// TIA Portal project "Controle_Por_Horario" (V18)

(* hardware
DEVICE "S7-1200 station_1"  S7-1200 Station
   slot 0: "Rack_0"  S7-1200 Rack  Rack  V1.0
   slot 1: "PLC_1"  CPU 1214C DC/DC/DC  6ES7 214-1AG40-0XB0  V4.5
DEVICE "HMI_1"  KTP700 Basic PN
   slot 0: "HMI_1"  KTP700 Basic PN  6AV2 123-2GB03-0AX0  17.0.0.0
   slot 1: "HMI_RT_1"  KTP700 Basic PN  6AV2 123-2GB03-0AX0  17.0.0.0
   slot 5: "HMI_1.IE_CP_1"  PROFINET Interface  17.0.0.0
      slot 1: "PROFINET Interface_1"  PROFINET Interface
         slot 1: "Port_1"  Port
*)

// ===== PLC "PLC_1"  CPU 1214C DC/DC/DC =====

VAR_GLOBAL   // PLC tag table "Default tag table"
   "System_Byte" AT %MB1 : Byte;
   "FirstScan" AT %M1.0 : Bool;
   "DiagStatusUpdate" AT %M1.1 : Bool;
   "AlwaysTRUE" AT %M1.2 : Bool;
   "AlwaysFALSE" AT %M1.3 : Bool;
   "Clock_Byte" AT %MB0 : Byte;
   "Clock_10Hz" AT %M0.0 : Bool;
   "Clock_5Hz" AT %M0.1 : Bool;
   "Clock_2.5Hz" AT %M0.2 : Bool;
   "Clock_2Hz" AT %M0.3 : Bool;
   "Clock_1.25Hz" AT %M0.4 : Bool;
   "Clock_1Hz" AT %M0.5 : Bool;
   "Clock_0.625Hz" AT %M0.6 : Bool;
   "Clock_0.5Hz" AT %M0.7 : Bool;
END_VAR

// folder: DBs

DATA_BLOCK "Var_IHM"   // DB1
{ S7_Optimized_Access := 'TRUE' }
VERSION : 0.1
   VAR
      Tela_Root : Struct
         Int_Date_Time_Local : Int;
         Date_Time_Formated : String;
         Date_Time : DTL;
         Bt_Liga_Habilita_Domingo : Bool;
         Bt_Liga_Habilita_Segunda : Bool;
         Bt_Liga_Habilita_Terca : Bool;
         Bt_Liga_Habilita_Quarta : Bool;
         Bt_Liga_Habilita_Quinta : Bool;
         Bt_Liga_Habilita_Sexta : Bool;
         Bt_Liga_Habilita_Sabado : Bool;
         Hora_Liga_Domingo : USInt;
         Minuto_Liga_Domingo : USInt;
         Hora_Liga_Segunda : USInt;
         Minuto_Liga_Segunda : USInt;
         Hora_Liga_Terca : USInt;
         Minuto_Liga_Terca : USInt;
         Hora_Liga_Quarta : USInt;
         Minuto_Liga_Quarta : USInt;
         Hora_Liga_Quinta : USInt;
         Minuto_Liga_Quinta : USInt;
         Hora_Liga_Sexta : USInt;
         Minuto_Liga_Sexta : USInt;
         Hora_Liga_Sabado : USInt;
         Minuto_Liga_Sabado : USInt;
         Hora_Desliga_Domingo : USInt;
         Minuto_Desliga_Domingo : USInt;
         Hora_Desliga_Segunda : USInt;
         Minuto_Desliga_Segunda : USInt;
         Hora_Desliga_Terca : USInt;
         Minuto_Desliga_Terca : USInt;
         Hora_Desliga_Quarta : USInt;
         Minuto_Desliga_Quarta : USInt;
         Hora_Desliga_Quinta : USInt;
         Minuto_Desliga_Quinta : USInt;
         Hora_Desliga_Sexta : USInt;
         Minuto_Desliga_Sexta : USInt;
         Hora_Desliga_Sabado : USInt;
         Minuto_Desliga_Sabado : USInt;
         Liga : Bool;
      END_STRUCT;
   END_VAR
BEGIN
END_DATA_BLOCK

// folder: (top level)

ORGANIZATION_BLOCK "Main"   // OB1, LAD, ProgramCycle
TITLE = "Main Program Sweep (Cycle)"
{ S7_Optimized_Access := 'TRUE' }
VERSION : 0.1
   VAR_INPUT
      Initial_Call : Bool;   // Initial call of this OB
      Remanence : Bool;   // =True, if remanent data are available
   END_VAR
BEGIN

REGION Network 1
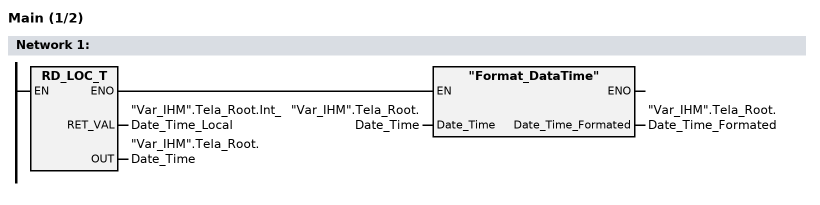
   // ENO of a box is taken as its EN; it also drops when the box reports an error
   "Var_IHM".Tela_Root.Int_Date_Time_Local := RD_LOC_T(OUT => "Var_IHM".Tela_Root.Date_Time);
   "Format_DataTime"(Date_Time := "Var_IHM".Tela_Root.Date_Time,
                     Date_Time_Formated => "Var_IHM".Tela_Root.Date_Time_Formated);
END_REGION

REGION Network 2
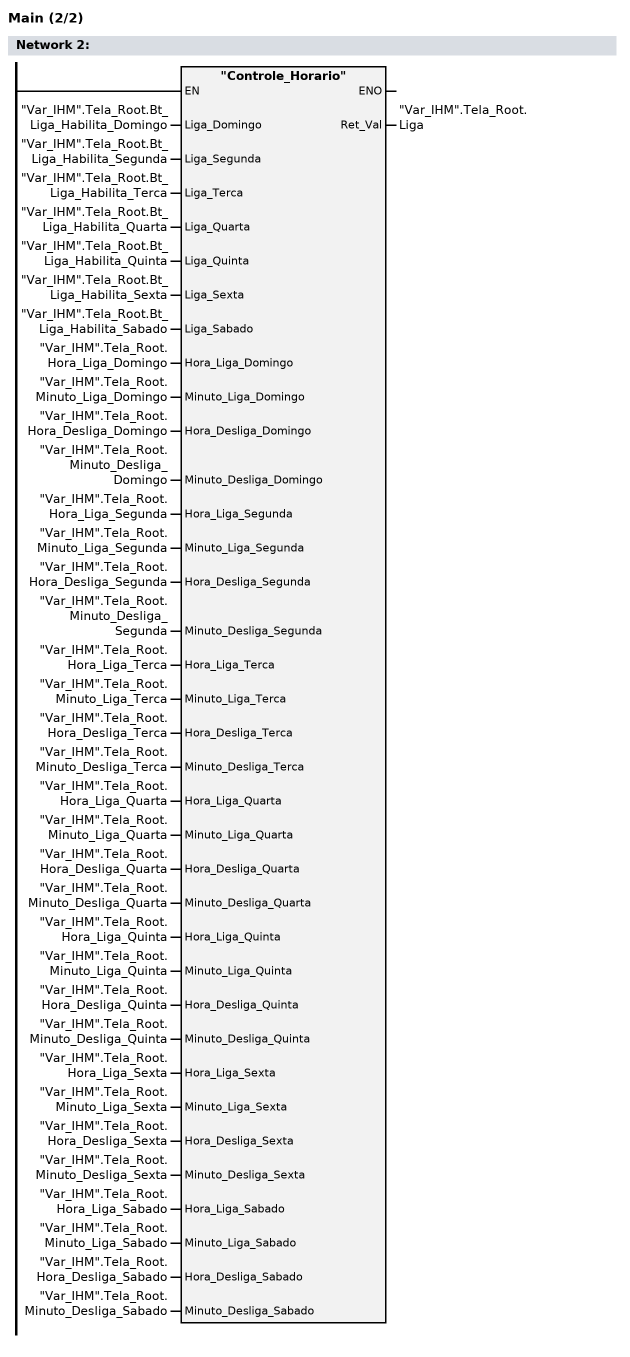
   RUNG wire#powerrail
      "Controle_Horario"(Liga_Domingo := "Var_IHM".Tela_Root.Bt_Liga_Habilita_Domingo, Liga_Segunda := "Var_IHM".Tela_Root.Bt_Liga_Habilita_Segunda, Liga_Terca := "Var_IHM".Tela_Root.Bt_Liga_Habilita_Terca, Liga_Quarta := "Var_IHM".Tela_Root.Bt_Liga_Habilita_Quarta, Liga_Quinta := "Var_IHM".Tela_Root.Bt_Liga_Habilita_Quinta, Liga_Sexta := "Var_IHM".Tela_Root.Bt_Liga_Habilita_Sexta, Liga_Sabado := "Var_IHM".Tela_Root.Bt_Liga_Habilita_Sabado, Hora_Liga_Domingo := "Var_IHM".Tela_Root.Hora_Liga_Domingo, Minuto_Liga_Domingo := "Var_IHM".Tela_Root.Minuto_Liga_Domingo, Hora_Desliga_Domingo := "Var_IHM".Tela_Root.Hora_Desliga_Domingo, Minuto_Desliga_Domingo := "Var_IHM".Tela_Root.Minuto_Desliga_Domingo, Hora_Liga_Segunda := "Var_IHM".Tela_Root.Hora_Liga_Segunda, Minuto_Liga_Segunda := "Var_IHM".Tela_Root.Minuto_Liga_Segunda, Hora_Desliga_Segunda := "Var_IHM".Tela_Root.Hora_Desliga_Segunda, Minuto_Desliga_Segunda := "Var_IHM".Tela_Root.Minuto_Desliga_Segunda, Hora_Liga_Terca := "Var_IHM".Tela_Root.Hora_Liga_Terca, Minuto_Liga_Terca := "Var_IHM".Tela_Root.Minuto_Liga_Terca, Hora_Desliga_Terca := "Var_IHM".Tela_Root.Hora_Desliga_Terca, Minuto_Desliga_Terca := "Var_IHM".Tela_Root.Minuto_Desliga_Terca, Hora_Liga_Quarta := "Var_IHM".Tela_Root.Hora_Liga_Quarta, Minuto_Liga_Quarta := "Var_IHM".Tela_Root.Minuto_Liga_Quarta, Hora_Desliga_Quarta := "Var_IHM".Tela_Root.Hora_Desliga_Quarta, Minuto_Desliga_Quarta := "Var_IHM".Tela_Root.Minuto_Desliga_Quarta, Hora_Liga_Quinta := "Var_IHM".Tela_Root.Hora_Liga_Quinta, Minuto_Liga_Quinta := "Var_IHM".Tela_Root.Minuto_Liga_Quinta, Hora_Desliga_Quinta := "Var_IHM".Tela_Root.Hora_Desliga_Quinta, Minuto_Desliga_Quinta := "Var_IHM".Tela_Root.Minuto_Desliga_Quinta, Hora_Liga_Sexta := "Var_IHM".Tela_Root.Hora_Liga_Sexta, Minuto_Liga_Sexta := "Var_IHM".Tela_Root.Minuto_Liga_Sexta, Hora_Desliga_Sexta := "Var_IHM".Tela_Root.Hora_Desliga_Sexta, Minuto_Desliga_Sexta := "Var_IHM".Tela_Root.Minuto_Desliga_Sexta, Hora_Liga_Sabado := "Var_IHM".Tela_Root.Hora_Liga_Sabado, Minuto_Liga_Sabado := "Var_IHM".Tela_Root.Minuto_Liga_Sabado, Hora_Desliga_Sabado := "Var_IHM".Tela_Root.Hora_Desliga_Sabado, Minuto_Desliga_Sabado := "Var_IHM".Tela_Root.Minuto_Desliga_Sabado, Ret_Val => "Var_IHM".Tela_Root.Liga)
   END_RUNG
   // the same network as SCL:
   "Var_IHM".Tela_Root.Liga := "Controle_Horario"(Liga_Domingo := "Var_IHM".Tela_Root.Bt_Liga_Habilita_Domingo,
                           Liga_Segunda := "Var_IHM".Tela_Root.Bt_Liga_Habilita_Segunda,
                           Liga_Terca := "Var_IHM".Tela_Root.Bt_Liga_Habilita_Terca,
                           Liga_Quarta := "Var_IHM".Tela_Root.Bt_Liga_Habilita_Quarta,
                           Liga_Quinta := "Var_IHM".Tela_Root.Bt_Liga_Habilita_Quinta,
                           Liga_Sexta := "Var_IHM".Tela_Root.Bt_Liga_Habilita_Sexta,
                           Liga_Sabado := "Var_IHM".Tela_Root.Bt_Liga_Habilita_Sabado,
                           Hora_Liga_Domingo := "Var_IHM".Tela_Root.Hora_Liga_Domingo,
                           Minuto_Liga_Domingo := "Var_IHM".Tela_Root.Minuto_Liga_Domingo,
                           Hora_Desliga_Domingo := "Var_IHM".Tela_Root.Hora_Desliga_Domingo,
                           Minuto_Desliga_Domingo := "Var_IHM".Tela_Root.Minuto_Desliga_Domingo,
                           Hora_Liga_Segunda := "Var_IHM".Tela_Root.Hora_Liga_Segunda,
                           Minuto_Liga_Segunda := "Var_IHM".Tela_Root.Minuto_Liga_Segunda,
                           Hora_Desliga_Segunda := "Var_IHM".Tela_Root.Hora_Desliga_Segunda,
                           Minuto_Desliga_Segunda := "Var_IHM".Tela_Root.Minuto_Desliga_Segunda,
                           Hora_Liga_Terca := "Var_IHM".Tela_Root.Hora_Liga_Terca,
                           Minuto_Liga_Terca := "Var_IHM".Tela_Root.Minuto_Liga_Terca,
                           Hora_Desliga_Terca := "Var_IHM".Tela_Root.Hora_Desliga_Terca,
                           Minuto_Desliga_Terca := "Var_IHM".Tela_Root.Minuto_Desliga_Terca,
                           Hora_Liga_Quarta := "Var_IHM".Tela_Root.Hora_Liga_Quarta,
                           Minuto_Liga_Quarta := "Var_IHM".Tela_Root.Minuto_Liga_Quarta,
                           Hora_Desliga_Quarta := "Var_IHM".Tela_Root.Hora_Desliga_Quarta,
                           Minuto_Desliga_Quarta := "Var_IHM".Tela_Root.Minuto_Desliga_Quarta,
                           Hora_Liga_Quinta := "Var_IHM".Tela_Root.Hora_Liga_Quinta,
                           Minuto_Liga_Quinta := "Var_IHM".Tela_Root.Minuto_Liga_Quinta,
                           Hora_Desliga_Quinta := "Var_IHM".Tela_Root.Hora_Desliga_Quinta,
                           Minuto_Desliga_Quinta := "Var_IHM".Tela_Root.Minuto_Desliga_Quinta,
                           Hora_Liga_Sexta := "Var_IHM".Tela_Root.Hora_Liga_Sexta,
                           Minuto_Liga_Sexta := "Var_IHM".Tela_Root.Minuto_Liga_Sexta,
                           Hora_Desliga_Sexta := "Var_IHM".Tela_Root.Hora_Desliga_Sexta,
                           Minuto_Desliga_Sexta := "Var_IHM".Tela_Root.Minuto_Desliga_Sexta,
                           Hora_Liga_Sabado := "Var_IHM".Tela_Root.Hora_Liga_Sabado,
                           Minuto_Liga_Sabado := "Var_IHM".Tela_Root.Minuto_Liga_Sabado,
                           Hora_Desliga_Sabado := "Var_IHM".Tela_Root.Hora_Desliga_Sabado,
                           Minuto_Desliga_Sabado := "Var_IHM".Tela_Root.Minuto_Desliga_Sabado);
END_REGION
END_ORGANIZATION_BLOCK

// folder: FCs

FUNCTION "Format_DataTime" : Void   // FC1, SCL
TITLE = Ezequiel
{ S7_Optimized_Access := 'TRUE' }
VERSION : 0.1
// Formata data e hora para o padrao DD/MM/YYYY  HH:MM:SS
   VAR_INPUT
      Date_Time : DTL;
   END_VAR
   VAR_OUTPUT
      Date_Time_Formated : String;
   END_VAR
   VAR_TEMP
      YEAR : String;
      MONTH : String;
      DAY : String;
      HOUR : String;
      MINUTE : String;
      SECOND : String;
      "DATE" : String;
      "TIME" : String;
   END_VAR
BEGIN
   #YEAR := UINT_TO_STRING(#Date_Time.YEAR);
   #YEAR := RIGHT(IN := #YEAR, L := 4);
   #MONTH := USINT_TO_STRING(#Date_Time.MONTH);

   IF #Date_Time.MONTH >= 10 THEN
       #MONTH := RIGHT(IN := #MONTH, L := 2);
   ELSE
       #MONTH := RIGHT(IN := #MONTH, L := 1);
       #MONTH := CONCAT(IN1 := '0', IN2 := #MONTH);
   END_IF;

   #DAY := USINT_TO_STRING(#Date_Time.DAY);

   IF #Date_Time.DAY >= 10 THEN
       #DAY := RIGHT(IN := #DAY, L := 2);
   ELSE
       #DAY := RIGHT(IN := #DAY, L := 1);
       #DAY := CONCAT(IN1 := '0', IN2 :=#DAY);
   END_IF;


   #HOUR := USINT_TO_STRING(#Date_Time.HOUR);

   IF #Date_Time.HOUR >= 10 THEN
       #HOUR := RIGHT(IN := #HOUR, L := 2);
   ELSE
       #HOUR := RIGHT(IN := #HOUR, L := 1);
   END_IF;

   #MINUTE := USINT_TO_STRING(#Date_Time.MINUTE);

   IF #Date_Time.MINUTE >= 10 THEN
       #MINUTE := RIGHT(IN := #MINUTE, L := 2);
   ELSE
       #MINUTE := RIGHT(IN := #MINUTE, L := 1);
       #MINUTE := CONCAT(IN1 := '0', IN2 := #MINUTE);
   END_IF;

   #SECOND := USINT_TO_STRING(#Date_Time.SECOND);

   IF #Date_Time.SECOND >= 10 THEN
       #SECOND := RIGHT(IN := #SECOND, L := 2);
   ELSE
       #SECOND := RIGHT(IN := #SECOND, L := 1);
       #SECOND := CONCAT(IN1 := '0', IN2 := #SECOND);
   END_IF;

   #DATE := CONCAT(IN1 := #DAY, IN2 := '/');
   #DATE := CONCAT(IN1 := #DATE, IN2 := #MONTH);
   #DATE := CONCAT(IN1 := #DATE, IN2 := '/');
   #DATE := CONCAT(IN1 := #DATE, IN2 := #YEAR);
   #DATE := CONCAT(IN1 := #DATE, IN2 := ' ');
   #TIME := CONCAT(IN1 := #HOUR, IN2 := ':');
   #TIME := CONCAT(IN1 := #TIME, IN2 := #MINUTE);
   #TIME := CONCAT(IN1 := #TIME, IN2 := ':');
   #TIME := CONCAT(IN1 := #TIME, IN2 := #SECOND);

   #Date_Time_Formated := CONCAT(IN1 := #DATE, IN2 := #TIME);
END_FUNCTION

FUNCTION "Controle_Horario" : Bool   // FC2, SCL
TITLE = FC de controle de horario
{ S7_Optimized_Access := 'TRUE' }
AUTHOR : Ezequiel
VERSION : 0.1
// FC habilita a saida conforme o dia da semana e horario programado
   VAR_INPUT
      Liga_Domingo : Bool;
      Liga_Segunda : Bool;
      Liga_Terca : Bool;
      Liga_Quarta : Bool;
      Liga_Quinta : Bool;
      Liga_Sexta : Bool;
      Liga_Sabado : Bool;
      Hora_Liga_Domingo : USInt;
      Minuto_Liga_Domingo : USInt;
      Hora_Desliga_Domingo : USInt;
      Minuto_Desliga_Domingo : USInt;
      Hora_Liga_Segunda : USInt;
      Minuto_Liga_Segunda : USInt;
      Hora_Desliga_Segunda : USInt;
      Minuto_Desliga_Segunda : USInt;
      Hora_Liga_Terca : USInt;
      Minuto_Liga_Terca : USInt;
      Hora_Desliga_Terca : USInt;
      Minuto_Desliga_Terca : USInt;
      Hora_Liga_Quarta : USInt;
      Minuto_Liga_Quarta : USInt;
      Hora_Desliga_Quarta : USInt;
      Minuto_Desliga_Quarta : USInt;
      Hora_Liga_Quinta : USInt;
      Minuto_Liga_Quinta : USInt;
      Hora_Desliga_Quinta : USInt;
      Minuto_Desliga_Quinta : USInt;
      Hora_Liga_Sexta : USInt;
      Minuto_Liga_Sexta : USInt;
      Hora_Desliga_Sexta : USInt;
      Minuto_Desliga_Sexta : USInt;
      Hora_Liga_Sabado : USInt;
      Minuto_Liga_Sabado : USInt;
      Hora_Desliga_Sabado : USInt;
      Minuto_Desliga_Sabado : USInt;
   END_VAR
   VAR_TEMP
      Data_Hora : DTL;
      Return_Data_Hora : Int;
      Ligou_Domingo : Bool;
      Ligou_Segunda : Bool;
      Ligou_Terca : Bool;
      Ligou_Quarta : Bool;
      Ligou_Quinta : Bool;
      Ligou_Sexta : Bool;
      Ligou_Sabado : Bool;
   END_VAR
BEGIN
   #Return_Data_Hora := RD_LOC_T(#Data_Hora);

   IF #Liga_Domingo AND #Data_Hora.WEEKDAY = 1 THEN
       IF (#Data_Hora.HOUR >= #Hora_Liga_Domingo AND #Data_Hora.MINUTE >= #Minuto_Liga_Domingo) THEN
           #Ligou_Domingo := TRUE;
       END_IF;
       IF (#Data_Hora.HOUR >= #Hora_Desliga_Domingo AND #Data_Hora.MINUTE >= #Minuto_Desliga_Domingo) THEN
           #Ligou_Domingo := FALSE;
       END_IF;
   END_IF;

   IF #Liga_Segunda AND #Data_Hora.WEEKDAY = 2 THEN
       IF (#Data_Hora.HOUR >= #Hora_Liga_Segunda AND #Data_Hora.MINUTE >= #Minuto_Liga_Segunda) THEN
           #Ligou_Segunda := TRUE;
       END_IF;
       IF (#Data_Hora.HOUR >= #Hora_Desliga_Segunda AND #Data_Hora.MINUTE >= #Minuto_Desliga_Segunda) THEN
           #Ligou_Segunda := FALSE;
       END_IF;
   END_IF;

   IF #Liga_Terca AND #Data_Hora.WEEKDAY = 3 THEN
       IF (#Data_Hora.HOUR >= #Hora_Liga_Terca AND #Data_Hora.MINUTE >= #Minuto_Liga_Terca) THEN
           #Ligou_Terca := TRUE;
       END_IF;
       IF (#Data_Hora.HOUR >= #Hora_Desliga_Terca AND #Data_Hora.MINUTE >= #Minuto_Desliga_Terca) THEN
           #Ligou_Terca := FALSE;
       END_IF;
   END_IF;

   IF #Liga_Quarta AND #Data_Hora.WEEKDAY = 4 THEN
       IF (#Data_Hora.HOUR >= #Hora_Liga_Quarta AND #Data_Hora.MINUTE >= #Minuto_Liga_Quarta) THEN
           #Ligou_Quarta := TRUE;
       END_IF;
       IF (#Data_Hora.HOUR >= #Hora_Desliga_Quarta AND #Data_Hora.MINUTE >= #Minuto_Desliga_Quarta) THEN
           #Ligou_Quarta := FALSE;
       END_IF;
   END_IF;

   IF #Liga_Quinta AND #Data_Hora.WEEKDAY = 5 THEN
       IF (#Data_Hora.HOUR >= #Hora_Liga_Quinta AND #Data_Hora.MINUTE >= #Minuto_Liga_Quinta) THEN
           #Ligou_Quinta := TRUE;
       END_IF;
       IF (#Data_Hora.HOUR >= #Hora_Desliga_Quinta AND #Data_Hora.MINUTE >= #Minuto_Desliga_Quinta) THEN
           #Ligou_Quinta := FALSE;
       END_IF;
   END_IF;

   IF #Liga_Sexta AND #Data_Hora.WEEKDAY = 6 THEN
       IF (#Data_Hora.HOUR >= #Hora_Liga_Sexta AND #Data_Hora.MINUTE >= #Minuto_Liga_Sexta) THEN
           #Ligou_Sexta := TRUE;
       END_IF;
       IF (#Data_Hora.HOUR >= #Hora_Desliga_Sexta AND #Data_Hora.MINUTE >= #Minuto_Desliga_Sexta) THEN
           #Ligou_Sexta := FALSE;
       END_IF;
   END_IF;

   IF #Liga_Sabado AND #Data_Hora.WEEKDAY = 7 THEN
       IF (#Data_Hora.HOUR >= #Hora_Liga_Sabado AND #Data_Hora.MINUTE >= #Minuto_Liga_Sabado) THEN
           #Ligou_Sabado := TRUE;
       END_IF;
       IF (#Data_Hora.HOUR >= #Hora_Desliga_Sabado AND #Data_Hora.MINUTE >= #Minuto_Desliga_Sabado) THEN
           #Ligou_Sabado := FALSE;
       END_IF;
   END_IF;

   #Controle_Horario := #Ligou_Domingo OR #Ligou_Segunda OR #Ligou_Terca OR #Ligou_Quarta OR #Ligou_Quinta OR #Ligou_Segunda OR #Ligou_Sabado;
END_FUNCTION

(* ===== HMI "HMI_RT_1" =====
system functions are stored by id; their names below are inferred from use
connection "HMI_Connection_1": ETHERNET, SMART_S7_1200_OMS

HMI tags "Default tag table"
   "Tag_ScreenNumber" : UInt, internal
   "Var_IHM_Tela_Root_Date_Time_Formated" : String[254] = PLC Var_IHM.Tela_Root.Date_Time_Formated, 1 s
   "Var_IHM_Tela_Root_Hora_Liga_Domingo" : USInt = PLC Var_IHM.Tela_Root.Hora_Liga_Domingo, 1 s
   "Var_IHM_Tela_Root_Hora_Liga_Segunda" : USInt = PLC Var_IHM.Tela_Root.Hora_Liga_Segunda, 1 s
   "Var_IHM_Tela_Root_Minuto_Liga_Domingo" : USInt = PLC Var_IHM.Tela_Root.Minuto_Liga_Domingo, 1 s
   "Var_IHM_Tela_Root_Minuto_Liga_Segunda" : USInt = PLC Var_IHM.Tela_Root.Minuto_Liga_Segunda, 1 s
   "Var_IHM_Tela_Root_Hora_Liga_Terca" : USInt = PLC Var_IHM.Tela_Root.Hora_Liga_Terca, 1 s
   "Var_IHM_Tela_Root_Minuto_Liga_Terca" : USInt = PLC Var_IHM.Tela_Root.Minuto_Liga_Terca, 1 s
   "Var_IHM_Tela_Root_Hora_Liga_Quarta" : USInt = PLC Var_IHM.Tela_Root.Hora_Liga_Quarta, 1 s
   "Var_IHM_Tela_Root_Minuto_Liga_Quarta" : USInt = PLC Var_IHM.Tela_Root.Minuto_Liga_Quarta, 1 s
   "Var_IHM_Tela_Root_Hora_Liga_Quinta" : USInt = PLC Var_IHM.Tela_Root.Hora_Liga_Quinta, 1 s
   "Var_IHM_Tela_Root_Minuto_Liga_Quinta" : USInt = PLC Var_IHM.Tela_Root.Minuto_Liga_Quinta, 1 s
   "Var_IHM_Tela_Root_Hora_Liga_Sexta" : USInt = PLC Var_IHM.Tela_Root.Hora_Liga_Sexta, 1 s
   "Var_IHM_Tela_Root_Minuto_Liga_Sexta" : USInt = PLC Var_IHM.Tela_Root.Minuto_Liga_Sexta, 1 s
   "Var_IHM_Tela_Root_Hora_Liga_Sabado" : USInt = PLC Var_IHM.Tela_Root.Hora_Liga_Sabado, 1 s
   "Var_IHM_Tela_Root_Minuto_Liga_Sabado" : USInt = PLC Var_IHM.Tela_Root.Minuto_Liga_Sabado, 1 s
   "Var_IHM_Tela_Root_Hora_Desliga_Domingo" : USInt = PLC Var_IHM.Tela_Root.Hora_Desliga_Domingo, 1 s
   "Var_IHM_Tela_Root_Minuto_Desliga_Domingo" : USInt = PLC Var_IHM.Tela_Root.Minuto_Desliga_Domingo, 1 s
   "Var_IHM_Tela_Root_Hora_Desliga_Segunda" : USInt = PLC Var_IHM.Tela_Root.Hora_Desliga_Segunda, 1 s
   "Var_IHM_Tela_Root_Hora_Desliga_Terca" : USInt = PLC Var_IHM.Tela_Root.Hora_Desliga_Terca, 1 s
   "Var_IHM_Tela_Root_Minuto_Desliga_Terca" : USInt = PLC Var_IHM.Tela_Root.Minuto_Desliga_Terca, 1 s
   "Var_IHM_Tela_Root_Hora_Desliga_Quarta" : USInt = PLC Var_IHM.Tela_Root.Hora_Desliga_Quarta, 1 s
   "Var_IHM_Tela_Root_Minuto_Desliga_Quarta" : USInt = PLC Var_IHM.Tela_Root.Minuto_Desliga_Quarta, 1 s
   "Var_IHM_Tela_Root_Hora_Desliga_Quinta" : USInt = PLC Var_IHM.Tela_Root.Hora_Desliga_Quinta, 1 s
   "Var_IHM_Tela_Root_Minuto_Desliga_Quinta" : USInt = PLC Var_IHM.Tela_Root.Minuto_Desliga_Quinta, 1 s
   "Var_IHM_Tela_Root_Hora_Desliga_Sexta" : USInt = PLC Var_IHM.Tela_Root.Hora_Desliga_Sexta, 1 s
   "Var_IHM_Tela_Root_Minuto_Desliga_Sexta" : USInt = PLC Var_IHM.Tela_Root.Minuto_Desliga_Sexta, 1 s
   "Var_IHM_Tela_Root_Hora_Desliga_Sabado" : USInt = PLC Var_IHM.Tela_Root.Hora_Desliga_Sabado, 1 s
   "Var_IHM_Tela_Root_Minuto_Desliga_Sabado" : USInt = PLC Var_IHM.Tela_Root.Minuto_Desliga_Sabado, 1 s
   "Var_IHM_Tela_Root_Bt_Liga_Habilita_Domingo" : Bool = PLC Var_IHM.Tela_Root.Bt_Liga_Habilita_Domingo, 1 s
   "Var_IHM_Tela_Root_Bt_Liga_Habilita_Segunda" : Bool = PLC Var_IHM.Tela_Root.Bt_Liga_Habilita_Segunda, 1 s
   "Var_IHM_Tela_Root_Bt_Liga_Habilita_Terca" : Bool = PLC Var_IHM.Tela_Root.Bt_Liga_Habilita_Terca, 1 s
   "Var_IHM_Tela_Root_Bt_Liga_Habilita_Quarta" : Bool = PLC Var_IHM.Tela_Root.Bt_Liga_Habilita_Quarta, 1 s
   "Var_IHM_Tela_Root_Bt_Liga_Habilita_Quinta" : Bool = PLC Var_IHM.Tela_Root.Bt_Liga_Habilita_Quinta, 1 s
   "Var_IHM_Tela_Root_Bt_Liga_Habilita_Sexta" : Bool = PLC Var_IHM.Tela_Root.Bt_Liga_Habilita_Sexta, 1 s
   "Var_IHM_Tela_Root_Bt_Liga_Habilita_Sabado" : Bool = PLC Var_IHM.Tela_Root.Bt_Liga_Habilita_Sabado, 1 s
   "Var_IHM_Tela_Root_Minuto_Desliga_Segunda" : USInt = PLC Var_IHM.Tela_Root.Minuto_Desliga_Segunda, 1 s
   "Var_IHM_Tela_Root_Liga" : Bool = PLC Var_IHM.Tela_Root.Liga, 1 s

Template "Template_1" 800x480
   Button "Alarms" at 714,429 size 71x50; TextOff 'Alarms'; PictureOff "AlarmDisplay_KTP700_Basic_PN_TR"; PictureOn "AlarmDisplay_KTP700_Basic_PN_TR"
      on Release: function_ef3f5d25("Alarm window_Unacknowledged", -1)
   Button "Template_Button" at 614,429 size 71x50; TextOff 'Text'
   Button "Template_Button_1" at 514,429 size 71x50; TextOff 'Text'
   Button "Template_Button_2" at 414,429 size 71x50; TextOff 'Text'
   Button "Template_Button_3" at 314,429 size 71x50; TextOff 'Text'
   Button "Template_Button_4" at 214,429 size 71x50; TextOff 'Text'
   Button "Template_Button_5" at 114,429 size 71x50; TextOff 'Text'
   Button "Start screen" at 14,429 size 71x50; TextOff 'Start screen'; PictureOff "NavigateHome_KTP700_Basic_PN_TR"; PictureOn "NavigateHome_KTP700_Basic_PN_TR"
      on Release: ActivateScreen("Root screen", 0)
   SymbolicIOField "Symbolic_IO_Field_Screen" at 93,9 size 600x33; TextOff '0'; TextOn '1'; TextList "TextList_ScreenNames"
      ProcessValue <- "Tag_ScreenNumber"
      on Change: ActivateScreenByNumber("Tag_ScreenNumber", 0)
   DateTimeField "HmiScreenItemData" at 695,25 size 105x25
   DateTimeField "HmiScreenItemData_1" at 695,0 size 105x25
   GraphicView "Logo" at 0,0 size 91x51; Picture "Logo of HMI_1"

screen "Root screen" 800x480, template "Template_1"
   on GenerateScreen: SetTag("Tag_ScreenNumber", 1)
   Button "HmiScreenItemData_1" at 17,49 size 159x47; TextOff 'System screens'; PictureOff "Navigates to System screens for KTP700 Basic+ PN 17.0.0.0"; PictureOn "Navigates to System screens for KTP700 Basic+ PN 17.0.0.0"
      on Release: ActivateScreen("System screens", 0)
   IOField "Template_I/O field_6" at 311,45 size 149x32; FormatPattern ????????????????????????????????????????
      ProcessValue <- "Var_IHM_Tela_Root_Date_Time_Formated"
   Switch "Switch_1" at 562,172 size 114x27; CaptionText 'Switch'; TextOff 'OFF'; TextOn 'ON'
      ProcessValue <- "Var_IHM_Tela_Root_Bt_Liga_Habilita_Domingo"
   IOField "I/O field_1" at 223,170 size 62x30; FormatPattern 99; Unit  Hrs
      ProcessValue <- "Var_IHM_Tela_Root_Hora_Liga_Domingo"
   TextField "Text field_1" at 129,174 size 77x23; Text 'Domingo'
   TextField "Text field_2" at 286,172 size 11x23; Text ':'
   IOField "I/O field_3" at 297,170 size 70x30; FormatPattern 99; Unit  min.
      ProcessValue <- "Var_IHM_Tela_Root_Minuto_Liga_Domingo"
   IOField "I/O field_2" at 396,170 size 62x30; FormatPattern 999; Unit  Hrs
      ProcessValue <- "Var_IHM_Tela_Root_Hora_Desliga_Domingo"
   TextField "Text field_3" at 459,172 size 11x23; Text ':'
   IOField "I/O field_4" at 470,170 size 70x30; FormatPattern 999; Unit  min.
      ProcessValue <- "Var_IHM_Tela_Root_Minuto_Desliga_Domingo"
   TextField "Text field_4" at 376,175 size 12x23; Text '-'
   Switch "Switch_2" at 562,207 size 114x27; TextOn 'ON'; CaptionText 'Switch'; TextOff 'OFF'
      ProcessValue <- "Var_IHM_Tela_Root_Bt_Liga_Habilita_Segunda"
   IOField "I/O field_5" at 223,205 size 62x30; FormatPattern 99; Unit  Hrs
      ProcessValue <- "Var_IHM_Tela_Root_Hora_Liga_Segunda"
   TextField "Text field_5" at 129,209 size 75x23; Text 'Segunda'
   TextField "Text field_6" at 286,207 size 11x23; Text ':'
   IOField "I/O field_6" at 297,205 size 70x30; FormatPattern 99; Unit  min.
      ProcessValue <- "Var_IHM_Tela_Root_Minuto_Liga_Segunda"
   IOField "I/O field_7" at 396,205 size 62x30; FormatPattern 999; Unit  Hrs
      ProcessValue <- "Var_IHM_Tela_Root_Hora_Desliga_Segunda"
   TextField "Text field_7" at 459,207 size 11x23; Text ':'
   IOField "I/O field_8" at 470,205 size 70x30; FormatPattern 999; Unit  min.
      ProcessValue <- "Var_IHM_Tela_Root_Minuto_Desliga_Segunda"
   TextField "Text field_8" at 376,210 size 12x23; Text '-'
   Switch "Switch_3" at 562,242 size 114x27; TextOn 'ON'; CaptionText 'Switch'; TextOff 'OFF'
      ProcessValue <- "Var_IHM_Tela_Root_Bt_Liga_Habilita_Terca"
   IOField "I/O field_9" at 223,240 size 62x30; FormatPattern 99; Unit  Hrs
      ProcessValue <- "Var_IHM_Tela_Root_Hora_Liga_Terca"
   TextField "Text field_9" at 129,244 size 51x23; Text 'Terça'
   TextField "Text field_10" at 286,242 size 11x23; Text ':'
   IOField "I/O field_10" at 297,240 size 70x30; FormatPattern 99; Unit  min.
      ProcessValue <- "Var_IHM_Tela_Root_Minuto_Liga_Terca"
   IOField "I/O field_11" at 396,240 size 62x30; FormatPattern 999; Unit  Hrs
      ProcessValue <- "Var_IHM_Tela_Root_Hora_Desliga_Terca"
   TextField "Text field_11" at 459,242 size 11x23; Text ':'
   IOField "I/O field_12" at 470,240 size 70x30; FormatPattern 999; Unit  min.
      ProcessValue <- "Var_IHM_Tela_Root_Minuto_Desliga_Terca"
   TextField "Text field_12" at 376,245 size 12x23; Text '-'
   Switch "Switch_4" at 562,277 size 114x27; TextOn 'ON'; CaptionText 'Switch'; TextOff 'OFF'
      ProcessValue <- "Var_IHM_Tela_Root_Bt_Liga_Habilita_Quarta"
   IOField "I/O field_13" at 223,275 size 62x30; FormatPattern 99; Unit  Hrs
      ProcessValue <- "Var_IHM_Tela_Root_Hora_Liga_Quarta"
   TextField "Text field_13" at 129,279 size 61x23; Text 'Quarta'
   TextField "Text field_14" at 286,277 size 11x23; Text ':'
   IOField "I/O field_14" at 297,275 size 70x30; FormatPattern 99; Unit  min.
      ProcessValue <- "Var_IHM_Tela_Root_Minuto_Liga_Quarta"
   IOField "I/O field_15" at 396,275 size 62x30; FormatPattern 999; Unit  Hrs
      ProcessValue <- "Var_IHM_Tela_Root_Hora_Desliga_Quarta"
   TextField "Text field_15" at 459,277 size 11x23; Text ':'
   IOField "I/O field_16" at 470,275 size 70x30; FormatPattern 999; Unit  min.
      ProcessValue <- "Var_IHM_Tela_Root_Minuto_Desliga_Quarta"
   TextField "Text field_16" at 376,280 size 12x23; Text '-'
   Switch "Switch_5" at 562,312 size 114x27; TextOn 'ON'; CaptionText 'Switch'; TextOff 'OFF'
      ProcessValue <- "Var_IHM_Tela_Root_Bt_Liga_Habilita_Quinta"
   IOField "I/O field_17" at 223,310 size 62x30; FormatPattern 99; Unit  Hrs
      ProcessValue <- "Var_IHM_Tela_Root_Hora_Liga_Quinta"
   TextField "Text field_17" at 129,314 size 59x23; Text 'Quinta'
   TextField "Text field_18" at 286,312 size 11x23; Text ':'
   IOField "I/O field_18" at 297,310 size 70x30; FormatPattern 99; Unit  min.
      ProcessValue <- "Var_IHM_Tela_Root_Minuto_Liga_Quinta"
   IOField "I/O field_19" at 396,310 size 62x30; FormatPattern 999; Unit  Hrs
      ProcessValue <- "Var_IHM_Tela_Root_Hora_Desliga_Quinta"
   TextField "Text field_19" at 459,312 size 11x23; Text ':'
   IOField "I/O field_20" at 470,310 size 70x30; FormatPattern 999; Unit  min.
      ProcessValue <- "Var_IHM_Tela_Root_Minuto_Desliga_Quinta"
   TextField "Text field_20" at 376,315 size 12x23; Text '-'
   Switch "Switch_6" at 562,347 size 114x27; TextOn 'ON'; CaptionText 'Switch'; TextOff 'OFF'
      ProcessValue <- "Var_IHM_Tela_Root_Bt_Liga_Habilita_Sexta"
   IOField "I/O field_21" at 223,345 size 62x30; FormatPattern 99; Unit  Hrs
      ProcessValue <- "Var_IHM_Tela_Root_Hora_Liga_Sexta"
   TextField "Text field_21" at 129,349 size 52x23; Text 'Sexta'
   TextField "Text field_22" at 286,347 size 11x23; Text ':'
   IOField "I/O field_22" at 297,345 size 70x30; FormatPattern 99; Unit  min.
      ProcessValue <- "Var_IHM_Tela_Root_Minuto_Liga_Sexta"
   IOField "I/O field_23" at 396,345 size 62x30; FormatPattern 999; Unit  Hrs
      ProcessValue <- "Var_IHM_Tela_Root_Hora_Desliga_Sexta"
   TextField "Text field_23" at 459,347 size 11x23; Text ':'
   IOField "I/O field_24" at 470,345 size 70x30; FormatPattern 999; Unit  min.
      ProcessValue <- "Var_IHM_Tela_Root_Minuto_Desliga_Sexta"
   TextField "Text field_24" at 376,350 size 12x23; Text '-'
   Switch "Switch_7" at 562,382 size 114x27; TextOn 'ON'; CaptionText 'Switch'; TextOff 'OFF'
      ProcessValue <- "Var_IHM_Tela_Root_Bt_Liga_Habilita_Sabado"
   IOField "I/O field_25" at 223,380 size 62x30; FormatPattern 99; Unit  Hrs
      ProcessValue <- "Var_IHM_Tela_Root_Hora_Liga_Sabado"
   TextField "Text field_25" at 129,384 size 65x23; Text 'Sábado'
   TextField "Text field_26" at 286,382 size 11x23; Text ':'
   IOField "I/O field_26" at 297,380 size 70x30; FormatPattern 99; Unit  min.
      ProcessValue <- "Var_IHM_Tela_Root_Minuto_Liga_Sabado"
   IOField "I/O field_27" at 396,380 size 62x30; FormatPattern 999; Unit  Hrs
      ProcessValue <- "Var_IHM_Tela_Root_Hora_Desliga_Sabado"
   TextField "Text field_27" at 459,382 size 11x23; Text ':'
   IOField "I/O field_28" at 470,380 size 70x30; FormatPattern 999; Unit  min.
      ProcessValue <- "Var_IHM_Tela_Root_Minuto_Desliga_Sabado"
   TextField "Text field_28" at 376,385 size 12x23; Text '-'
   TextField "Text field_29" at 269,133 size 39x23; Text 'Liga'
   TextField "Text field_30" at 431,133 size 65x23; Text 'Desliga'
   Circle "Circle_1" at 429,89 size 30x30
      Appearance <- "Var_IHM_Tela_Root_Liga"
   TextField "Text field_31" at 339,93 size 76x23; Text 'Liberado'

screen "System screens" 800x480, template "Template_1"
   on GenerateScreen: SetTag("Tag_ScreenNumber", 2)
   Button "Back" at 1,52 size 159x47; TextOff 'Back'
      on Release: ActivateScreen("Root screen", 0)
   Button "HmiScreenItemData" at 36,146 size 159x47; TextOff 'SIMATIC PLC system diagnos...'; PictureOff "Navigates to SIMATIC PLC system diagnostics for KTP700 Basic+ PN 17.0.0.0"; PictureOn "Navigates to SIMATIC PLC system diagnostics for KTP700 Basic+ PN 17.0.0.0"
      on Release: ActivateScreen("SIMATIC PLC system diagnostics", 0)
   Button "HmiScreenItemData_1" at 36,205 size 159x47; TextOff 'Project information'; PictureOff "Navigates to Project information for KTP700 Basic+ PN 17.0.0.0"; PictureOn "Navigates to Project information for KTP700 Basic+ PN 17.0.0.0"
      on Release: ActivateScreen("Project information", 0)
   Button "HmiScreenItemData_2" at 36,264 size 159x47; TextOff 'User administration'; PictureOff "Navigates to User administration for KTP700 Basic+ PN 17.0.0.0"; PictureOn "Navigates to User administration for KTP700 Basic+ PN 17.0.0.0"
      on Release: ActivateScreen("User administration", 0)
   Button "HmiScreenItemData_3" at 36,323 size 159x47; TextOff 'System information'; PictureOff "Navigates to System information for KTP700 Basic+ PN 17.0.0.0"; PictureOn "Navigates to System information for KTP700 Basic+ PN 17.0.0.0"
      on Release: ActivateScreen("System information", 0)

screen "SIMATIC PLC system diagnostics" 800x480, template "Template_1"
   on GenerateScreen: SetTag("Tag_ScreenNumber", 3)
   SysDiagControl "HmiScreenItemData" at 1,100 size 796x321
   Button "Back" at 1,52 size 159x47; TextOff 'Back'
      on Release: ActivateScreen("System screens", 0)

screen "Project information" 800x480, template "Template_1"
   on GenerateScreen: SetTag("Tag_ScreenNumber", 4)
   TextField "HmiScreenItemData" at 35,102 size 171x28; Text 'Project name:'
   TextField "HmiScreenItemData_1" at 241,102 size 524x28; Text 'Format_Time'
   TextField "HmiScreenItemData_2" at 35,132 size 171x28; Text 'Created on:'
   TextField "HmiScreenItemData_3" at 241,132 size 524x28; Text '8/29/2024 8:20:00 AM'
   TextField "HmiScreenItemData_4" at 35,162 size 171x28; Text 'Author:'
   TextField "HmiScreenItemData_5" at 241,162 size 524x28; Text 'Ezequiel'
   TextField "HmiScreenItemData_6" at 35,192 size 171x28; Text 'Description:'
   TextField "HmiScreenItemData_7" at 241,192 size 524x28; Text '(not configured)'
   Button "Back" at 1,52 size 159x47; TextOff 'Back'
      on Release: ActivateScreen("System screens", 0)

screen "User administration" 800x480, template "Template_1"
   on GenerateScreen: SetTag("Tag_ScreenNumber", 5)
   UserView "HmiScreenItemData" at 1,100 size 796x321
   Button "Back" at 1,52 size 159x47; TextOff 'Back'
      on Release: ActivateScreen("System screens", 0)

screen "System information" 800x480, template "Template_1"
   on GenerateScreen: SetTag("Tag_ScreenNumber", 6)
   TextField "HmiScreenItemData" at 35,102 size 171x28; Text 'HMI device type:'
   TextField "HmiScreenItemData_1" at 241,102 size 524x28; Text 'KTP700 Basic+ PN 17.0.0.0'
   TextField "HmiScreenItemData_2" at 35,132 size 171x28; Text 'Connection:'
   TextField "HmiScreenItemData_3" at 241,132 size 524x28; Text 'PROFINET (X1)'
   TextField "HmiScreenItemData_4" at 35,162 size 171x28; Text 'PLC:'
   TextField "HmiScreenItemData_5" at 241,162 size 524x28; Text 'SIMATIC S7 1200'
   Button "Back" at 1,52 size 159x47; TextOff 'Back'
      on Release: ActivateScreen("System screens", 0)
*)